FUNCTION F_InRange : BOOL
VAR_INPUT
    value 		: LREAL;
    lower_limit : LREAL;
    upper_limit : LREAL;
END_VAR
VAR
END_VAR

F_InRange := (lower_limit <= value) AND (value <= upper_limit);

END_FUNCTION

(* stored: Version 1.1.0.1, ProductVersion 3.1.4024.12
   POU F_InRange: Id {4657ece0-e5a2-4b60-99c7-98cbe76d1b78}, SpecialFunc None *)
